TYPE "TokenChain_Data"
VERSION : 0.1
// Block: TokenChain_Data
   STRUCT
      TOKEN : Int;
      USER : Int;
      OldToken : Int;
      TimeOut : IEC_TIMER;
   END_STRUCT;

END_TYPE
